// TIA Portal V19 export
TYPE "LAF_typeHeaderHmiToPlc"
// Information from the HMI to the PLC
// stored: Access Published
   STRUCT
      acknowledge : Bool;   // Acknowledge command
      powerCommands : Byte;   // On/Off command
      selectedUnits : Word := 16#01;   // Selected units from the HMI
      modeRequests : Word;   // Mode requested recieved from the HMI
      stateCommands : Word;   // State command recieved from the HMI
      specialFunctions : Word;   // Special functions recieved from the HMI
   END_STRUCT;
END_TYPE
